FUNCTION_BLOCK ABSTRACT Heating_State EXTENDS State
VAR
	_ctx			: REFERENCE TO Heating_Ctx;
END_VAR

(*FB_Init is always available implicitly and it is used primarily for initialization.
The return value is not evaluated. For a specific influence, you can also declare the
methods explicitly and provide additional code there with the standard initialization
code. You can evaluate the return value.*)
METHOD FB_Init : BOOL
VAR_INPUT
	(* TRUE: the retain variables are initialized (reset warm / reset cold)*)
	bInitRetains	: BOOL;
	(* TRUE: the instance will be copied to the copy code afterward (online change)*)
	bInCopyCode	: BOOL;
	iEntity	: Core.I_Entity;
	ctx		: REFERENCE TO Heating_Ctx;
END_VAR
_ctx REF= ctx;
END_METHOD

END_FUNCTION_BLOCK

(* stored: Version 1.1.0.1
   POU Heating_State: Id {3fb4f9bd-5291-4ac7-ba56-d4e8ec1876e7}, SpecialFunc None
   Method FB_Init: Id {627f5069-2cda-4b66-b3cc-d02d905db010} *)
